// TIA Portal V20 export
DATA_BLOCK "GRIP_TUNE"   // DB67
{ S7_Optimized_Access := 'FALSE' }
VERSION : 0.1
// stored: AutoNumber true, DBAccessibleFromOPCUA true, DBAccessibleFromWebserver true, IsOnlyStoredInLoadMemory false, IsWriteProtectedInAS false
   VAR
      Tune { S7_SetPoint := 'True'} : "LGR_GripperTune";   // FB_CL_Gripper 학습 · 보정값. 표준 접근 : gr-console 이 읽고 (ScaleByInch 는) 쓴다
   END_VAR
BEGIN
END_DATA_BLOCK
